{attribute 'GeneratedUsingTerminal: EK1100-0000-0018'}
{attribute addProperty BoxType "EK1100-0000-0018"}
{attribute addProperty Id "Beckhoff_EPP3xxxEK1122Beckhoff_EPP3xxxEK1122_56CB9FB31280"}
{attribute addProperty CRC "1794246294"}
{attribute addProperty Size "1280"}
TYPE Beckhoff_EPP3xxx_6AF20696 EXTENDS EK1100_1FC0878B :
STRUCT
	{attribute addProperty Name "Beckhoff_EPP3xxxEK1122"}
	{attribute addProperty PreviousPort "Beckhoff EPP3xxx : B"}
	Beckhoff_EPP3xxxEK1122 : Beckhoff_EPP3xxxEK1122_56CB9FB3;
END_STRUCT
END_TYPE

(* stored: Version 1.2.0.0, ProductVersion 3.1.4024.9
   DUT Beckhoff_EPP3xxx_6AF20696: Id {3b0d5d50-23ce-4886-8b38-3810c7c4c50a} *)
